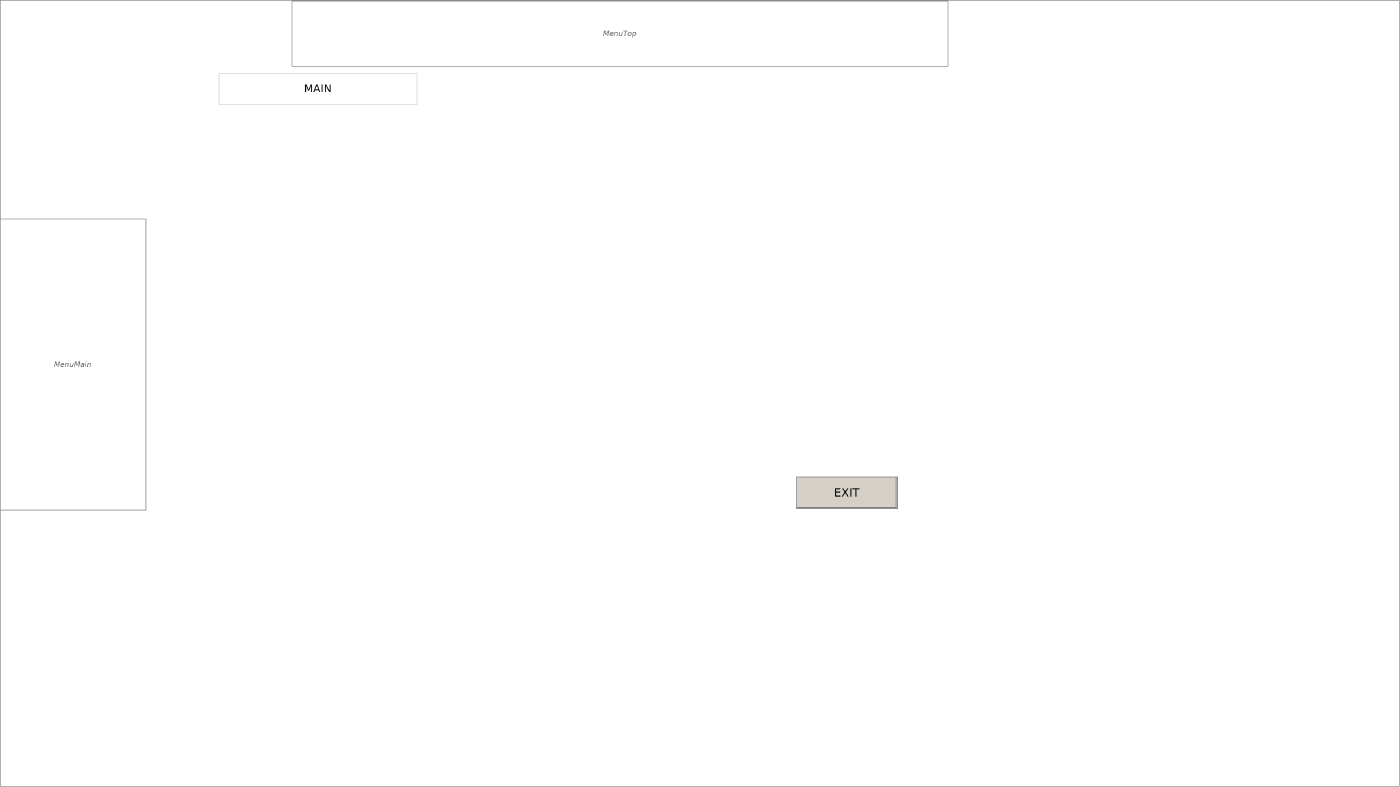
VISUALIZATION MainScreen  // 1920x1080
    Frame (400,1 900x90)
        shows MenuTop()
    Frame (0,300 200x400)
        shows MenuMain()
    Textfield (300,100 272x43), "MAIN"
    Button (1092,654 139x44), "EXIT"
        OnMouseClick: ExecuteCommand ExecuteCommand=ExecuteCommand=[Command=ExecuteClientProgram, Value='TASKKILL /F /IM', Value2='Tc3PlcHmi.exe']
END_VISUALIZATION

(* stored: Version 1.1.0.1, ProductVersion 3.1.4024.10
   Visu MainScreen: Id {db7d3618-78e0-4151-89b4-068b857ba3ef} *)
